Staubli VAL3: deleteItem.pgx

public program deleteItem(num x_nIndex, num& x_nResult[])
  local num l_nFound
  local num l_nSize
  local num i
  local InstrItem l_sEvent
begin
  //
  // delete the selected field
  //
  call getSizeItem(l_nSize)
  l_nFound=0
  for i=0 to (l_nSize-1)
    call getItem(l_sEvent,i)
    if find(l_sEvent.sType,"#")!=-1
      l_nFound=-1
      call delEvent(i)
      i=i-1
      call getSizeItem(l_nSize)
    endIf
  endFor
  //
  // if there are no marked events delete the select one
  //
  if x_nIndex!=-1 and l_nFound==0
    call delEvent(x_nIndex)
  endIf
end
